// TIA Portal project "GR36_BP_BeltConveyorGreen_Transport1xBox" (V17)

(* hardware
DEVICE "S7-1200 station_1"  S7-1200 Station
   slot 0: "Rack_0"  S7-1200 Rack  Rack  V1.0
   slot 1: "PLC_1"  CPU 1214C DC/DC/DC  6ES7 214-1AG31-0XB0  V3.0
*)

// ===== PLC "PLC_1"  CPU 1214C DC/DC/DC =====

VAR_GLOBAL   // PLC tag table "math"
   "mb_a1" AT %MB130 : SInt;
   "mb_a2" AT %MB131 : SInt;
   "mb_aResult" AT %MW132 : Int;
   "mb_b1" AT %MB136 : SInt;
   "md_b2" AT %MD138 : DInt;
   "mb_c1" AT %MB146 : SInt;
   "mb_c2" AT %MB147 : SInt;
   "mw_cResult" AT %MW148 : Int;
   "md_bResult" AT %MD142 : DInt;
   "mw_d1" AT %MW150 : Int;
   "mw_d2" AT %MW152 : Int;
   "md_dResult" AT %MD154 : DInt;
   "mb_e1" AT %MB158 : SInt;
   "mb_e2" AT %MB159 : SInt;
   "md_eResult" AT %MD160 : Real;
   "mw_RPM" AT %MW164 : Int;
   "mw_Gear" AT %MW166 : Int;
   "mw_DiameterShaft_mm" AT %MW168 : Int;
   "md_SpeedBelt_mm_s" AT %MD170 : Real;
END_VAR

VAR_GLOBAL   // PLC tag table "MemoryFlag_PLC"
   "m_IsAutoModeForwardRunning" AT %M0.0 : Bool;
END_VAR

VAR_GLOBAL   // PLC tag table "DigitalOutput_PLC"
   "dq_LedGreen" AT %Q4.0 : Bool;
   "dq_LedRed" AT %Q4.1 : Bool;
   "dq_LedWhite" AT %Q4.2 : Bool;
   "dq_LedBlue" AT %Q4.3 : Bool;
   "dq_Horn" AT %Q4.4 : Bool;
   "dqb_Lights" AT %QB4 : Byte;
END_VAR

VAR_GLOBAL   // PLC tag table "DigitalInput_PLC"
   "di_Switch_Forward" AT %I1.4 : Bool;   // NO
   "di_Switch_Backward" AT %I1.5 : Bool;   // NO
   "di_Switch_SwitchBay1" AT %I1.6 : Bool;   // NO
   "di_Switch_SwitchBay2" AT %I1.7 : Bool;   // NO
   "di_StartButton" AT %I2.0 : Bool;   // NO
   "di_StopButton" AT %I2.1 : Bool;   // NC
   "di_Selector" AT %I2.2 : Bool;   // NO
   "di_ResetButton" AT %I2.3 : Bool;   // NC
   "dib_switch" AT %IB1 : Byte;
END_VAR

VAR_GLOBAL   // PLC tag table "DigitalOutput_FactoryIO"
   "dq_Forward" AT %Q0.0 : Bool;
   "dq_Backward" AT %Q0.1 : Bool;
END_VAR

VAR_GLOBAL   // PLC tag table "DigitalInput_FactoryIO"
   "di_AtLeft_B0" AT %I0.0 : Bool;   // NO
   "di_AtMiddle_B3" AT %I0.1 : Bool;   // NC
   "di_AtRight_B5" AT %I0.2 : Bool;   // NO
   "di_FactoryIO_Running" AT %I0.7 : Bool;
   "di_ImpulsFromShaft" AT %I0.5 : Bool;
END_VAR

VAR_GLOBAL   // PLC tag table "DefultTagTable"
   "Clock_Byte" AT %MB69 : Byte;
   "Clock_10Hz" AT %M69.0 : Bool;
   "Clock_5Hz" AT %M69.1 : Bool;
   "Clock_2.5Hz" AT %M69.2 : Bool;
   "Clock_2Hz" AT %M69.3 : Bool;
   "Clock_1.25Hz" AT %M69.4 : Bool;
   "Clock_1Hz" AT %M69.5 : Bool;
   "Clock_0.625Hz" AT %M69.6 : Bool;
   "Clock_0.5Hz" AT %M69.7 : Bool;
   "System_Byte" AT %MB70 : Byte;
   "FirstScan" AT %M70.0 : Bool;
   "DiagStatusUpdate" AT %M70.1 : Bool;
   "AlwaysTRUE" AT %M70.2 : Bool;
   "AlwaysFALSE" AT %M70.3 : Bool;
   "System_Byte(1)" AT %MB1 : Byte;
   "Tag_1" AT %M10.0 : Bool;
   "Tag_2" AT %M10.1 : Bool;
   "Tag_3" AT %M20.0 : Bool;
   "Tag_4" AT %M20.7 : Bool;
   "Tag_5" AT %M21.2 : Bool;
   "Tag_6" AT %MB120 : USInt;
   "Tag_7" AT %M120.1 : Bool;
   "Tag_8" AT %M255.0 : Bool;
   "Tag_9" AT %M255.1 : Bool;
   "Tag_10" AT %M255.7 : Bool;
   "Tag_11" AT %M255.4 : Bool;
   "Tag_12" AT %M266.0 : Bool;
   "Tag_13" AT %M170.2 : Bool;
END_VAR

VAR_GLOBAL   // PLC tag table "Default tag table"
   "Tag_14" AT %M120.0 : Bool;
END_VAR

DATA_BLOCK "db_Output"   // DB1
{ S7_Optimized_Access := 'TRUE' }
VERSION : 0.1
   VAR
      Forward_Manual : Bool;
      Forward_Auto : Bool;
      Backward_Manual : Bool;
      Backward_Auto : Bool;
   END_VAR
BEGIN
END_DATA_BLOCK

DATA_BLOCK "db_Mode"   // DB2
{ S7_Optimized_Access := 'TRUE' }
VERSION : 0.1
   VAR
      Manual : Bool;
      Auto : Bool;
      GlobalError : Bool;
   END_VAR
BEGIN
END_DATA_BLOCK

DATA_BLOCK "db_Error"   // DB3
{ S7_Optimized_Access := 'TRUE' }
VERSION : 0.1
   VAR
      ID0_TimeOut : Bool := 0;
      ID1 : Bool;
   END_VAR
BEGIN
END_DATA_BLOCK

DATA_BLOCK "db_Settings"   // DB4
{ S7_Optimized_Access := 'TRUE' }
VERSION : 0.1
   VAR RETAIN
      WatiForStart : Time := T#2s;
      MaxTransportTime : Time := T#14s;
   END_VAR
   VAR
      DelayWithdrawFromLine : Time := t#2s;
   END_VAR
BEGIN
END_DATA_BLOCK

// folder: System blocks/Program resources

DATA_BLOCK "TON_DelayForwardAuto"   // DB5
{ S7_Optimized_Access := 'TRUE' }
AUTHOR : Simatic
FAMILY : IEC
NAME : IEC_TMR
VERSION : 1.0
// stored: InstanceOfName IEC_TIMER
"IEC_TIMER"
BEGIN
END_DATA_BLOCK

DATA_BLOCK "TON_ErrorTimeout"   // DB6
{ S7_Optimized_Access := 'TRUE' }
AUTHOR : Simatic
FAMILY : IEC
NAME : IEC_TMR
VERSION : 1.0
// stored: InstanceOfName IEC_TIMER
"IEC_TIMER"
BEGIN
END_DATA_BLOCK

DATA_BLOCK "TP_DelayWitchdrawFromConveyor"   // DB7
{ S7_Optimized_Access := 'TRUE' }
AUTHOR : Simatic
FAMILY : IEC
NAME : IEC_TMR
VERSION : 1.0
// stored: InstanceOfName IEC_TIMER
"IEC_TIMER"
BEGIN
END_DATA_BLOCK

// folder: (top level)

FUNCTION "FC_Mode" : Void   // FC1, LAD
{ S7_Optimized_Access := 'TRUE' }
VERSION : 0.1
BEGIN

REGION Network 1: Handle Maunal Mode
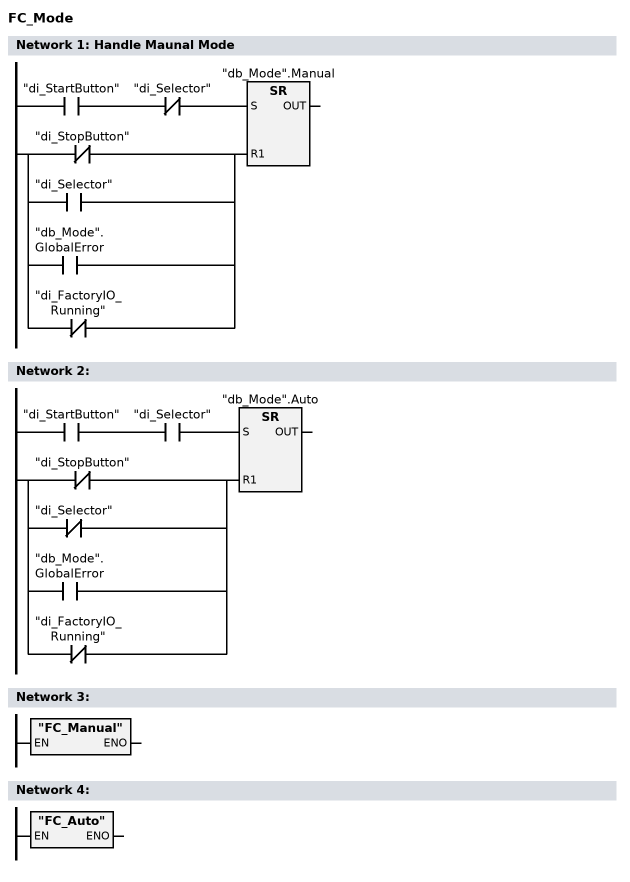
   RUNG wire#powerrail
      Contact( "di_StartButton" )
      I_Contact( "di_Selector" )
      S_SR(operand := "db_Mode".Manual, r1 := wire#w1)
   END_RUNG
   RUNG wire#powerrail
      I_Contact( "di_StopButton" )
   END_RUNG wire#w1
   RUNG wire#powerrail
      Contact( "di_Selector" )
   END_RUNG wire#w1
   RUNG wire#powerrail
      Contact( "db_Mode".GlobalError )
   END_RUNG wire#w1
   RUNG wire#powerrail
      I_Contact( "di_FactoryIO_Running" )
   END_RUNG wire#w1
   // the same network as SCL:
   IF "di_StartButton" AND NOT "di_Selector" THEN
       "db_Mode".Manual := TRUE;   // SR flip-flop
   END_IF;
   IF NOT "di_StopButton" OR "di_Selector" OR "db_Mode".GlobalError OR NOT "di_FactoryIO_Running" THEN
       "db_Mode".Manual := FALSE;
   END_IF;
END_REGION

REGION Network 2
   RUNG wire#powerrail
      Contact( "di_StartButton" )
      Contact( "di_Selector" )
      S_SR(operand := "db_Mode".Auto, r1 := wire#w1)
   END_RUNG
   RUNG wire#powerrail
      I_Contact( "di_StopButton" )
   END_RUNG wire#w1
   RUNG wire#powerrail
      I_Contact( "di_Selector" )
   END_RUNG wire#w1
   RUNG wire#powerrail
      Contact( "db_Mode".GlobalError )
   END_RUNG wire#w1
   RUNG wire#powerrail
      I_Contact( "di_FactoryIO_Running" )
   END_RUNG wire#w1
   // the same network as SCL:
   IF "di_StartButton" AND "di_Selector" THEN
       "db_Mode".Auto := TRUE;   // SR flip-flop
   END_IF;
   IF NOT "di_StopButton" OR NOT "di_Selector" OR "db_Mode".GlobalError OR NOT "di_FactoryIO_Running" THEN
       "db_Mode".Auto := FALSE;
   END_IF;
END_REGION

REGION Network 3
   RUNG wire#powerrail
      "FC_Manual"()
   END_RUNG
   // the same network as SCL:
   "FC_Manual"();
END_REGION

REGION Network 4
   RUNG wire#powerrail
      "FC_Auto"()
   END_RUNG
   // the same network as SCL:
   "FC_Auto"();
END_REGION
END_FUNCTION

FUNCTION "FC_Manual" : Void   // FC2, LAD
{ S7_Optimized_Access := 'TRUE' }
VERSION : 0.1
BEGIN

REGION Network 1
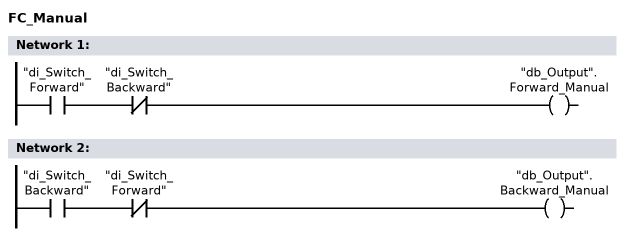
   RUNG wire#powerrail
      Contact( "di_Switch_Forward" )
      I_Contact( "di_Switch_Backward" )
      Coil( "db_Output".Forward_Manual )
   END_RUNG
   // the same network as SCL:
   "db_Output".Forward_Manual := "di_Switch_Forward" AND NOT "di_Switch_Backward";
END_REGION

REGION Network 2
   RUNG wire#powerrail
      Contact( "di_Switch_Backward" )
      I_Contact( "di_Switch_Forward" )
      Coil( "db_Output".Backward_Manual )
   END_RUNG
   // the same network as SCL:
   "db_Output".Backward_Manual := "di_Switch_Backward" AND NOT "di_Switch_Forward";
END_REGION
END_FUNCTION

FUNCTION "FC_Auto" : Void   // FC3, LAD
{ S7_Optimized_Access := 'TRUE' }
VERSION : 0.1
   VAR_TEMP   // added for the SCL form of the ladder/FBD networks
      _w1 : Bool;
   END_VAR
BEGIN

REGION Network 1: Auto Mode
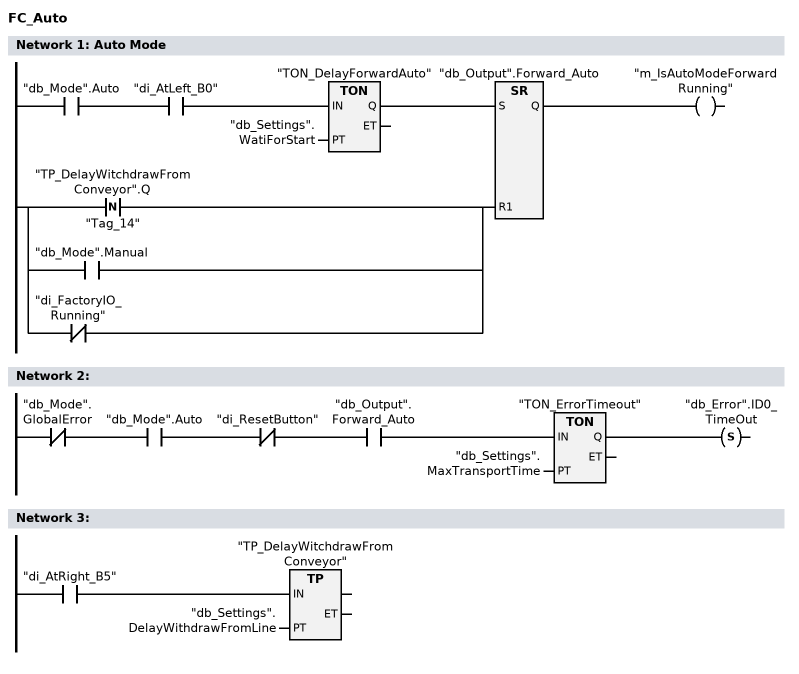
   "TON_DelayForwardAuto".TON(IN := "db_Mode".Auto AND "di_AtLeft_B0", PT := "db_Settings".WatiForStart);
   #_w1 := NOT "TP_DelayWitchdrawFromConveyor".Q AND "Tag_14";   // falling edge of "TP_DelayWitchdrawFromConveyor".Q
   "Tag_14" := "TP_DelayWitchdrawFromConveyor".Q;
   IF "TON_DelayForwardAuto".Q THEN
       "db_Output".Forward_Auto := TRUE;   // SR flip-flop
   END_IF;
   IF #_w1 OR "db_Mode".Manual OR NOT "di_FactoryIO_Running" THEN "db_Output".Forward_Auto := FALSE; END_IF;
   "m_IsAutoModeForwardRunning" := "db_Output".Forward_Auto;
END_REGION

REGION Network 2
   "TON_ErrorTimeout".TON(IN := NOT "db_Mode".GlobalError AND "db_Mode".Auto AND NOT "di_ResetButton" AND "db_Output".Forward_Auto,
                          PT := "db_Settings".MaxTransportTime);
   IF "TON_ErrorTimeout".Q THEN "db_Error".ID0_TimeOut := TRUE; END_IF;
END_REGION

REGION Network 3
   "TP_DelayWitchdrawFromConveyor".TP(IN := "di_AtRight_B5", PT := "db_Settings".DelayWithdrawFromLine);
END_REGION
END_FUNCTION

FUNCTION "FC_LightSygnalization" : Void   // FC4, LAD
{ S7_Optimized_Access := 'TRUE' }
VERSION : 0.1
BEGIN

REGION Network 1
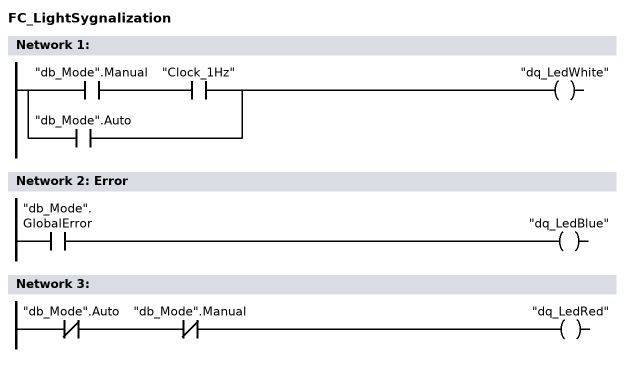
   RUNG wire#powerrail
      Contact( "db_Mode".Manual )
      Contact( "Clock_1Hz" )
      wire#w1
      Coil( "dq_LedWhite" )
   END_RUNG
   RUNG wire#powerrail
      Contact( "db_Mode".Auto )
   END_RUNG wire#w1
   // the same network as SCL:
   "dq_LedWhite" := ("db_Mode".Manual AND "Clock_1Hz") OR "db_Mode".Auto;
END_REGION

REGION Network 2: Error
   RUNG wire#powerrail
      Contact( "db_Mode".GlobalError )
      Coil( "dq_LedBlue" )
   END_RUNG
   // the same network as SCL:
   "dq_LedBlue" := "db_Mode".GlobalError;
END_REGION

REGION Network 3
   RUNG wire#powerrail
      I_Contact( "db_Mode".Auto )
      I_Contact( "db_Mode".Manual )
      Coil( "dq_LedRed" )
   END_RUNG
   // the same network as SCL:
   "dq_LedRed" := NOT "db_Mode".Auto AND NOT "db_Mode".Manual;
END_REGION
END_FUNCTION

FUNCTION "FC_Output" : Void   // FC5, LAD
{ S7_Optimized_Access := 'TRUE' }
VERSION : 0.1
BEGIN

REGION Network 1: Forward
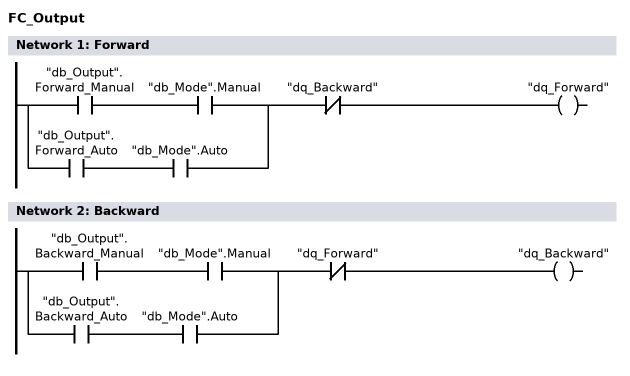
   RUNG wire#powerrail
      Contact( "db_Output".Forward_Manual )
      Contact( "db_Mode".Manual )
      wire#w1
      I_Contact( "dq_Backward" )
      Coil( "dq_Forward" )
   END_RUNG
   RUNG wire#powerrail
      Contact( "db_Output".Forward_Auto )
      Contact( "db_Mode".Auto )
   END_RUNG wire#w1
   // the same network as SCL:
   "dq_Forward" := (("db_Output".Forward_Manual AND "db_Mode".Manual) OR ("db_Output".Forward_Auto AND "db_Mode".Auto)) AND NOT "dq_Backward";
END_REGION

REGION Network 2: Backward
   RUNG wire#powerrail
      Contact( "db_Output".Backward_Manual )
      Contact( "db_Mode".Manual )
      wire#w1
      I_Contact( "dq_Forward" )
      Coil( "dq_Backward" )
   END_RUNG
   RUNG wire#powerrail
      Contact( "db_Output".Backward_Auto )
      Contact( "db_Mode".Auto )
   END_RUNG wire#w1
   // the same network as SCL:
   "dq_Backward" := (("db_Output".Backward_Manual AND "db_Mode".Manual) OR ("db_Output".Backward_Auto AND "db_Mode".Auto)) AND NOT "dq_Forward";
END_REGION
END_FUNCTION

FUNCTION "FC_Error" : Void   // FC6, LAD
{ S7_Optimized_Access := 'TRUE' }
VERSION : 0.1
BEGIN

REGION Network 1
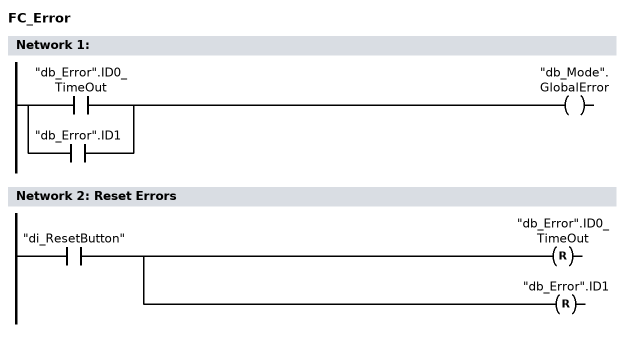
   RUNG wire#powerrail
      Contact( "db_Error".ID0_TimeOut )
      wire#w1
      Coil( "db_Mode".GlobalError )
   END_RUNG
   RUNG wire#powerrail
      Contact( "db_Error".ID1 )
   END_RUNG wire#w1
   // the same network as SCL:
   "db_Mode".GlobalError := "db_Error".ID0_TimeOut OR "db_Error".ID1;
END_REGION

REGION Network 2: Reset Errors
   RUNG wire#powerrail
      Contact( "di_ResetButton" )
      wire#w1
      R_Coil( "db_Error".ID0_TimeOut )
   END_RUNG
   RUNG wire#w1
      R_Coil( "db_Error".ID1 )
   END_RUNG
   // the same network as SCL:
   IF "di_ResetButton" THEN
       "db_Error".ID0_TimeOut := FALSE;
       "db_Error".ID1 := FALSE;
   END_IF;
END_REGION
END_FUNCTION

ORGANIZATION_BLOCK "Main"   // OB1, LAD, ProgramCycle
TITLE = "Main Program Sweep (Cycle)"
{ S7_Optimized_Access := 'TRUE' }
VERSION : 0.1
BEGIN

REGION Network 1
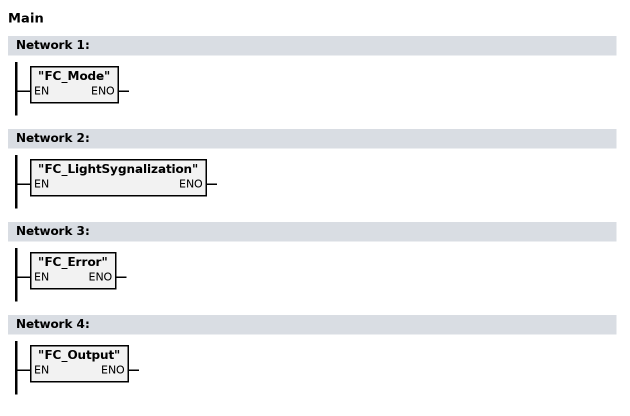
   RUNG wire#powerrail
      "FC_Mode"()
   END_RUNG
   // the same network as SCL:
   "FC_Mode"();
END_REGION

REGION Network 2
   RUNG wire#powerrail
      "FC_LightSygnalization"()
   END_RUNG
   // the same network as SCL:
   "FC_LightSygnalization"();
END_REGION

REGION Network 3
   RUNG wire#powerrail
      "FC_Error"()
   END_RUNG
   // the same network as SCL:
   "FC_Error"();
END_REGION

REGION Network 4
   RUNG wire#powerrail
      "FC_Output"()
   END_RUNG
   // the same network as SCL:
   "FC_Output"();
END_REGION
END_ORGANIZATION_BLOCK